Omron CX-Programmer project NewProject (CX-Programmer 9.03)

# PLC NewPLC1: CJ1M CPU11
I/O table (CPU CJ1M-CPU11): rack 0 slot 0 CJ1W-ETN21(ETN11Mode); rack 0 slot 1 CJ1W-ID211; rack 0 slot 2 CJ1W-OD211; rack 0 slot 3 CJ1W-ID211; rack 0 slot 4 CJ1W-OD211; rack 0 slot 5 CJ1W-ID211; rack 0 slot 6 CJ1W-OD232

## Program NewProgram1 (cyclic task 0)
Local symbols
B1 1.04 BOOL
Cond W0.01 BOOL
Eletro1 1.06 BOOL
Eletro2 1.07 BOOL
Eletro3 1.08 BOOL
Eletro4 1.09 BOOL
M1 1.00 BOOL
M2 1.01 BOOL
M3 1.02 BOOL
M4 1.03 BOOL
Sensor1 0.00 BOOL
Sensor2 0.01 BOOL
Sensor3 0.02 BOOL
Sensor4 0.03 BOOL
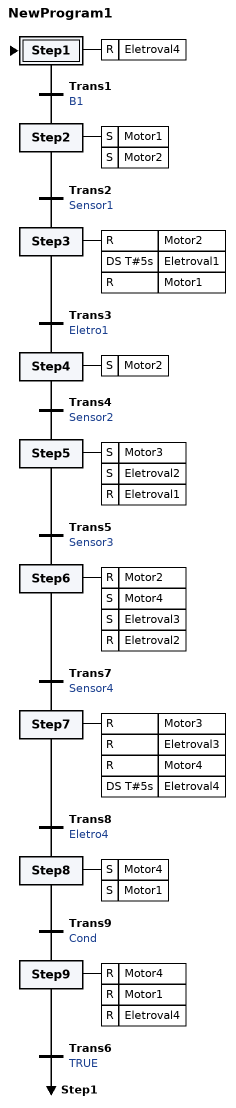
INITIAL_STEP Step1 :
Eletroval4(R) ;
END_STEP
TRANSITION Trans1 FROM Step1 TO Step2
 := B1;
END_TRANSITION
STEP Step2 :
Motor1(S) ;
Motor2(S) ;
END_STEP
TRANSITION Trans2 FROM Step2 TO Step3
 := Sensor1;
END_TRANSITION
STEP Step3 :
Motor2(R) ;
Eletroval1(DS,T#5s) ;
Motor1(R) ;
END_STEP
TRANSITION Trans3 FROM Step3 TO Step4
 := Eletro1;
END_TRANSITION
STEP Step4 :
Motor2(S) ;
END_STEP
TRANSITION Trans4 FROM Step4 TO Step5
 := Sensor2;
END_TRANSITION
STEP Step5 :
Motor3(S) ;
Eletroval2(S) ;
Eletroval1(R) ;
END_STEP
TRANSITION Trans5 FROM Step5 TO Step6
 := Sensor3;
END_TRANSITION
STEP Step6 :
Motor2(R) ;
Motor4(S) ;
Eletroval3(S) ;
Eletroval2(R) ;
END_STEP
TRANSITION Trans6 FROM Step9 TO Step1
 := TRUE;
END_TRANSITION
TRANSITION Trans7 FROM Step6 TO Step7
 := Sensor4;
END_TRANSITION
STEP Step7 :
Motor3(R) ;
Eletroval3(R) ;
Motor4(R) ;
Eletroval4(DS,T#5s) ;
END_STEP
TRANSITION Trans8 FROM Step7 TO Step8
 := Eletro4;
END_TRANSITION
STEP Step8 :
Motor4(S) ;
Motor1(S) ;
END_STEP
TRANSITION Trans9 FROM Step8 TO Step9
 := Cond;
END_TRANSITION
STEP Step9 :
Motor4(R) ;
Motor1(R) ;
Eletroval4(R) ;
END_STEP

### Action Motor1

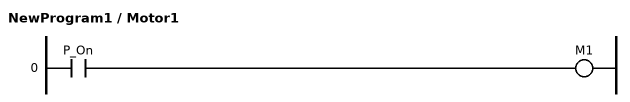
; rung 0
LD P_On
OUT M1

### Action Motor2

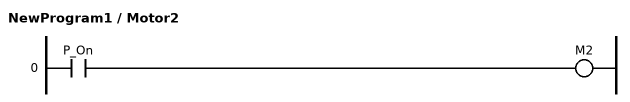
; rung 0
LD P_On
OUT M2

### Action Eletroval1

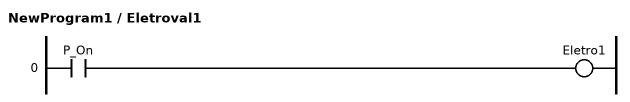
; rung 0
LD P_On
OUT Eletro1

### Action Eletroval2

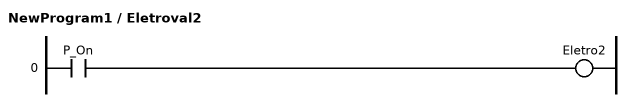
; rung 0
LD P_On
OUT Eletro2

### Action Eletroval3

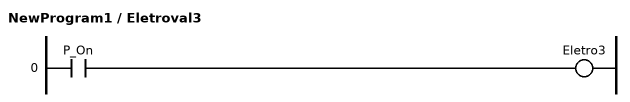
; rung 0
LD P_On
OUT Eletro3

### Action Eletroval4

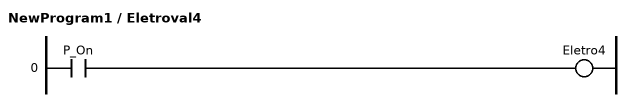
; rung 0
LD P_On
OUT Eletro4

### Action Motor3

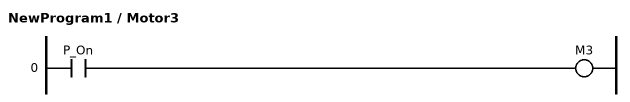
; rung 0
LD P_On
OUT M3

### Action Motor4

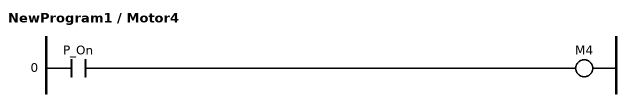
; rung 0
LD P_On
OUT M4